// TIA Portal project "cobotTry" (V19)

(* hardware
DEVICE "S7-1200 station_1"  S7-1200 Station
   slot 0: "Rack_0"  S7-1200 Rack  Rack  V1.0
   slot 1: "PLC_1"  CPU 1214C AC/DC/Rly  6ES7 214-1BG40-0XB0  V4.5
   slot 2: "DI 16x24VDC/DQ 16xRelay_1"  SM 1223 DI16/DQ16 x relay  6ES7 223-1PL32-0XB0  V2.0
   slot 3: "AI 4x13BIT/AQ 2x14BIT_1"  6ES7 234-4HE32-0XB0  V2.1
   slot 3: "AQ 1x12BIT_1"  AQ1 signal board  6ES7 232-4HA30-0XB0  V1.0
*)

// ===== PLC "PLC_1"  CPU 1214C AC/DC/Rly =====

VAR_GLOBAL   // PLC tag table "Default tag table"
   "Tag_1" AT %M10.0 : Bool;
   "Tag_2" AT %M10.1 : Bool;
   "Tag_3" AT %M10.2 : Bool;
   "Tag_4" AT %Q8.1 : Bool;
   "Tag_5" AT %Q8.2 : Bool;
   "Tag_6" AT %Q9.4 : Bool;
   "Tag_7" AT %I0.1 : Bool;
   "Tag_8" AT %I0.2 : Bool;
   "Tag_9" AT %M10.3 : Bool;
   "Tag_10" AT %M10.4 : Bool;
   "Tag_11" AT %M10.5 : Bool;
END_VAR

ORGANIZATION_BLOCK "Main"   // OB1, LAD, ProgramCycle
TITLE = "Main Program Sweep (Cycle)"
{ S7_Optimized_Access := 'TRUE' }
VERSION : 0.1
   VAR_INPUT
      Initial_Call : Bool;   // Initial call of this OB
      Remanence : Bool;   // =True, if remanent data are available
   END_VAR
BEGIN

REGION Network 1
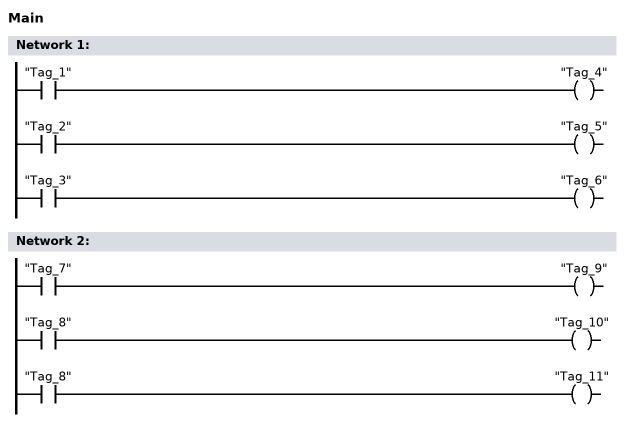
   RUNG wire#powerrail
      Contact( "Tag_1" )
      Coil( "Tag_4" )
   END_RUNG
   RUNG wire#powerrail
      Contact( "Tag_2" )
      Coil( "Tag_5" )
   END_RUNG
   RUNG wire#powerrail
      Contact( "Tag_3" )
      Coil( "Tag_6" )
   END_RUNG
   // the same network as SCL:
   "Tag_4" := "Tag_1";
   "Tag_5" := "Tag_2";
   "Tag_6" := "Tag_3";
END_REGION

REGION Network 2
   RUNG wire#powerrail
      Contact( "Tag_7" )
      Coil( "Tag_9" )
   END_RUNG
   RUNG wire#powerrail
      Contact( "Tag_8" )
      Coil( "Tag_10" )
   END_RUNG
   RUNG wire#powerrail
      Contact( "Tag_8" )
      Coil( "Tag_11" )
   END_RUNG
   // the same network as SCL:
   "Tag_9" := "Tag_7";
   "Tag_10" := "Tag_8";
   "Tag_11" := "Tag_8";
END_REGION
END_ORGANIZATION_BLOCK